(* CoDeSys 2.3.9.62 project: Practica1Ej2.pro *)

(* Global variable list: Global_Variables *)
VAR_GLOBAL
  (* Entradas *)
	A: BOOL;
	B: BOOL;
(* Salidas *)
	salrojo: BOOL;
       salverde:BOOL;

END_VAR

(* POU PLC_PRG, FBD *)
PROGRAM PLC_PRG
VAR

END_VAR
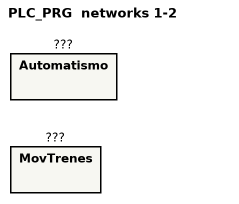
_FBD_ (* Function Block Diagram *)
NETWORK 1
	???:Automatismo()
NETWORK 2
	???:MovTrenes()
_END_FBD_
END_PROGRAM

(* POU Automatismo, LD *)
PROGRAM Automatismo
VAR

	E0: BOOL;
	E1: BOOL;
	E2: BOOL;
	SA: BOOL;
	SB: BOOL;
END_VAR
VAR (* helpers for the ST form of the networks *)
	_p1 : BOOL;
	_p2 : BOOL;
	_p3 : BOOL;
END_VAR
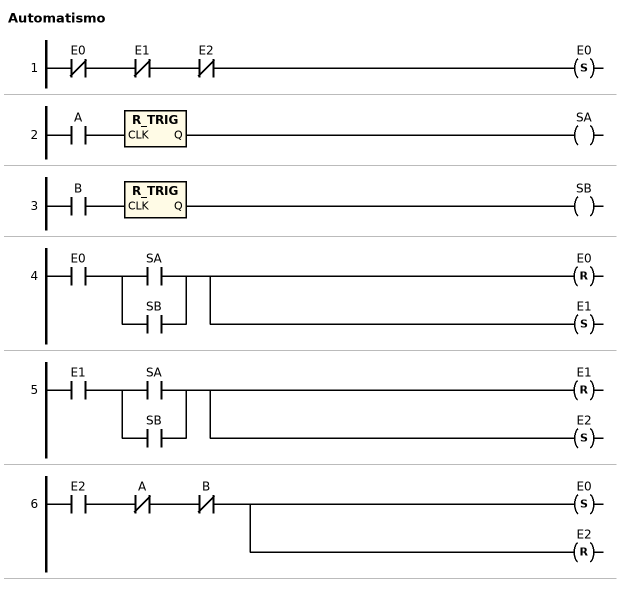
_LD_ (* Ladder Diagram *)
NETWORK 1
	[/E0] - [/E1] - [/E2] --- (S E0)
NETWORK 2
	[A] - R_TRIG(CLK: *) --- (SA)
NETWORK 3
	[B] - R_TRIG(CLK: *) --- (SB)
NETWORK 4
	[E0] - { [SA] | [SB] } --- (R E0) (S E1)
NETWORK 5
	[E1] - { [SA] | [SB] } --- (R E1) (S E2)
NETWORK 6
	[E2] - [/A] - [/B] --- (S E0) (R E2)
_END_LD_
(* the same logic as Structured Text *)
(* Network 1 *)
IF NOT E0 AND NOT E1 AND NOT E2 THEN E0 := TRUE; END_IF;
(* Network 2 *)
SA := R_TRIG(CLK := A);
(* Network 3 *)
SB := R_TRIG(CLK := B);
(* Network 4 *)
_p1 := E0 AND (SA OR SB);
IF _p1 THEN E0 := FALSE; E1 := TRUE; END_IF;
(* Network 5 *)
_p2 := E1 AND (SA OR SB);
IF _p2 THEN E1 := FALSE; E2 := TRUE; END_IF;
(* Network 6 *)
_p3 := E2 AND NOT A AND NOT B;
IF _p3 THEN E0 := TRUE; E2 := FALSE; END_IF;
END_PROGRAM

(* POU MovTrenes, ST *)
PROGRAM MovTrenes
VAR
  ENTRA_IZQ:BOOL;
	tren_izq: BOOL;
	posx: INT :=-550;
	ENTRA_DER: BOOL;
	tren_der: BOOL;
       vel:INT;
END_VAR
IF (ENTRA_IZQ=TRUE) AND (tren_der=FALSE) THEN
    tren_izq:=TRUE;
ELSE
   IF  (ENTRA_DER=TRUE) AND (tren_izq=FALSE) AND (tren_der=FALSE) THEN
       tren_der:=TRUE;
      posx:=390;
   END_IF
END_IF

IF (tren_izq=TRUE) THEN
   posx:=posx+2+vel;
END_IF


IF (tren_der=TRUE) THEN
   posx:=posx-2-vel;
END_IF

IF (posx>-430) AND (posx<-100) THEN
   A:=TRUE;
ELSE
   A:=FALSE;
END_IF

IF (posx>16) AND (posx<350) THEN
   B:=TRUE;
ELSE
   B:=FALSE;
END_IF

IF (posx>400) AND (tren_izq=TRUE)  THEN
    tren_izq:=FALSE;
    posx:=-550;
END_IF


IF (posx<-500) AND (tren_der=TRUE) THEN
    tren_der:=FALSE;
    posx:=-550;
END_IF
END_PROGRAM

(* Visualisation Tren
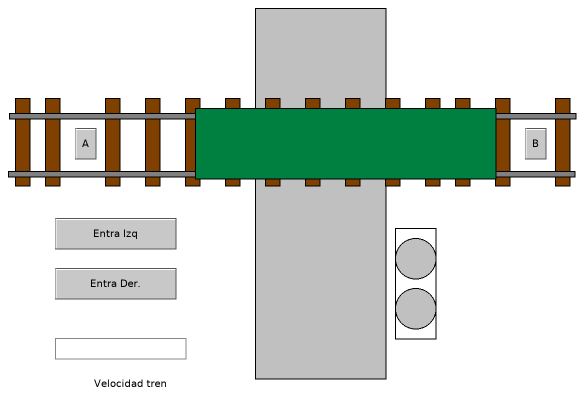
button at (60,120)-(81,151): text "A"; toggles A
button at (510,120)-(531,151): text "B"; toggles B
ellipse at (380,230)-(421,271): alarm colour if salrojo
ellipse at (380,280)-(421,321): alarm colour if salverde
rounded rectangle at (180,100)-(481,171): x offset MovTrenes.posx
button at (40,210)-(161,241): text "Entra Izq"; taps MovTrenes.ENTRA_IZQ
button at (40,260)-(161,291): text "Entra Der."; taps MovTrenes.ENTRA_DER
rectangle at (30,360)-(201,391): text "Velocidad tren"
19 more shapes without text or variables
*)
